FUNCTION MeasureUnit_to_EngUnits : REAL
VAR_INPUT
	rValue		: REAL;
	rSlope 		: REAL;
	rOffset 	: REAL;
END_VAR
VAR
END_VAR

MeasureUnit_to_EngUnits := (rValue*rSlope)+rOffset;

END_FUNCTION

(* stored: Version 1.1.0.1, ProductVersion 3.1.4024.12
   POU MeasureUnit_to_EngUnits: Id {9f488d98-284d-4172-b00e-a49132af1263}, SpecialFunc None *)
